VAR_GLOBAL
	
//lichtsturing
LichtenRAAMKANT AT %Q*: BOOL;
LichtenDEURKANT AT %Q*: BOOL;

AanwezigheidsdetectorRAAMKANT AT %I*: BOOL;
AanwezigheidsdetectorDEURKANT AT %I*: BOOL;

LichtsterkteDEUR AT %I*: INT;
LichtsterkteDEUR2 AT %I*: INT;
LichtsterkteBORD AT %I*: INT;
lichtsterkteBORD2 AT %I*: INT;
LINKERKNOP AT %I* : BOOL;
RECHTERKNOP AT %I* : BOOL;


//beamer & projectorschermsturing

BeamerAANKNOP AT %I* : BOOL;
BeamerUITKNOP AT %I* : BOOL;
Projectorscherm AT %Q* : BOOL;



socketconnectknop AT %I* : BOOL;
socketsendknop AT %I* : BOOL;



//raamsturing


stKL6581            : STR_KL6581;


//Lora
	sDatastring: STRING(500);
	
	Moteeui			: STRING;
	Appeui			: STRING;
	UserData		: ST_UserData;
	PayloadDecoded	: STRING;

	PayloadLength	: DINT;
	PayloadData		: ARRAY[1..100] OF BYTE;
	NullByte		: BYTE := 0;


END_VAR

(* stored: Version 1.1.0.1, ProductVersion 3.1.4022.10
   GVL GVL1: Id {812b4598-46c3-4a6c-843c-c938bd265cfd} *)
